FUNCTION_BLOCK FB_Members EXTENDS FB_ListComponent implements I_Members
VAR_INPUT
END_VAR
VAR_OUTPUT
END_VAR
VAR
END_VAR

METHOD PUBLIC M_Abort : BOOL (* Return state complete*)

VAR
	nIndex: DINT;
END_VAR
M_Abort:= TRUE;
WHILE nIndex < nLength DO
	IF M_Index(nIndex).M_RequestState(E_RequestState.Abort) THEN
		;
	ELSE
		M_Abort:= FALSE;
	END_IF

	nIndex:= nIndex + 1;
END_WHILE
END_METHOD

METHOD PUBLIC M_Attach : BOOL
VAR_INPUT
	iParent:	I_Component;
	iObject: 	I_Component;
END_VAR
M_Add(iObject);
iObject.P_Event.P_Logger:= iParent.P_Event.P_Logger;
iObject.P_Event.P_Observer.M_Attach(iParent);
M_Attach:= True;
END_METHOD

METHOD PUBLIC M_Detach : BOOL
VAR_INPUT
	iParent:	I_Component;
	iObject: 	I_Component;
END_VAR
M_Remove(iObject);
iObject.P_Event.P_Logger:= 0;
iObject.P_Event.P_Observer.M_Detach(iParent);
M_Detach:= True;
END_METHOD

{attribute 'TcRpcEnable':='1'}
METHOD PUBLIC M_Mode : BOOL
VAR_INPUT
	eMode:		E_RequestMode;
END_VAR

VAR
	nIndex: DINT;
END_VAR
WHILE nIndex < nLength DO
	M_Index(nIndex).M_RequestMode(eMode);
	nIndex:= nIndex + 1;
END_WHILE
M_Mode:= TRUE;
END_METHOD

METHOD PUBLIC M_Reset : BOOL

VAR
	nIndex: DINT;
END_VAR
WHILE nIndex < nLength DO
	M_Index(nIndex).M_RequestState(E_RequestState.Reset);
	nIndex:= nIndex + 1;
END_WHILE
M_Reset:= TRUE;
END_METHOD

METHOD PUBLIC M_Start : BOOL (* Return state complete*)

VAR
	nIndex: DINT;
END_VAR
M_Start:= TRUE;
WHILE nIndex < nLength DO
	IF M_Index(nIndex).M_RequestState(E_RequestState.Start) THEN
		;
	ELSE
		M_Start:= FALSE;
	END_IF
	
	nIndex:= nIndex + 1;
END_WHILE
END_METHOD

METHOD PUBLIC M_Stop : BOOL (* Return state complete*)

VAR
	nIndex: DINT;
END_VAR
M_Stop:= TRUE;
WHILE nIndex < nLength DO
	IF M_Index(nIndex).M_RequestState(E_RequestState.Stop) THEN
		;
	ELSE
		M_Stop:= FALSE;
	END_IF

	nIndex:= nIndex + 1;
END_WHILE
END_METHOD

END_FUNCTION_BLOCK

(* stored: Version 1.1.0.1
   POU FB_Members: Id {cd8da5ab-5393-0aad-280e-8aa1aa48dea2}, SpecialFunc None
   Method M_Abort: Id {ca242ed0-a742-02fd-2f25-ec86a9ce81af}
   Method M_Attach: Id {f766bba5-1031-00ce-2c1e-fef5e99d9284}
   Method M_Detach: Id {a6e34f01-76bf-0e93-0f6e-f335e6f09f85}
   Method M_Mode: Id {06622676-d17f-00c9-0303-c4ed42551906}
   Method M_Reset: Id {f82c528d-d106-0d47-26b7-c180584df544}
   Method M_Start: Id {ae13c90b-3cbf-07f6-16fc-7e76ef730bbf}
   Method M_Stop: Id {e019d36a-59f9-03ae-0272-fef9a290f8db} *)
